{attribute 'GeneratedUsingTerminal: EK1122-0000-0018'}
{attribute addProperty BoxType "EK1122-0000-0018"}
{attribute addProperty Id "Beckhoff_EM2xxxsub_EK1100EK1100_1FC0878B2"}
{attribute addProperty CRC "3082833217"}
{attribute addProperty Size "2"}
TYPE Beckhoff_EM2xxxEK1122_B7C04D41 EXTENDS EK1122_1FC0878B :
STRUCT
	{attribute addProperty Name "Beckhoff EM2xxxsub EK1100"}
	{attribute addProperty PreviousPort "Beckhoff EM2xxxEK1122 : D"}
	Beckhoff_EM2xxxsub_EK1100 : EK1100_1FC0878B;
END_STRUCT
END_TYPE
